{attribute addProperty BoxType "EL9210-0000-0016"}
{attribute addProperty Id "PowerOKAT %I*BOOL81"}
{attribute addProperty CRC "1532743738"}
{attribute addProperty SizeInBites "8"}
{attribute addProperty SizeInBytes "1"}
TYPE PowerOK_5B5BD03A :
STRUCT
	{attribute addProperty Name "PowerOK"}
	PowerOK AT %I* : BOOL;
END_STRUCT
END_TYPE

(* stored: Version 1.2.0.0, ProductVersion 3.1.4024.9
   DUT PowerOK_5B5BD03A: Id {0d7b73f3-4d41-49a8-80a3-8de802a7c065} *)
